FUNCTION_BLOCK FB_SmartMotor
VAR_INPUT
END_VAR
VAR_OUTPUT
END_VAR
VAR
	nStartCount : INT :=0;
END_VAR

METHOD Counter : INT
VAR_INPUT
END_VAR
nStartCount := nStartCount + 1;
END_METHOD

END_FUNCTION_BLOCK

(* stored: Version 1.1.0.1, ProductVersion 3.1.4024.16
   POU FB_SmartMotor: Id {d78028df-126f-4a98-b687-5e01347f9090}, SpecialFunc None
   Method Counter: Id {61cc2fe1-d7a6-4838-84e5-63ccccb76962} *)
